FUNCTION_BLOCK FB_XPlanarModule EXTENDS FB_PackML_BaseModule
VAR
	// Component definitions here
	XPlanarTable : FB_Component_Xplanar := (Name := 'XPlanarTable');

	//Station Components
	Station1 : FB_RotateStation := (Name := 'Station1'); //Declaration of a custom station
	Station2 : FB_TiltStation := (Name := 'Station2');
	Station3 : FB_BounceStation := (Name := 'Station3');

	//Helper Vars
	Mover			  : ARRAY[1..SystemParameters.MOVER_COUNT] OF FB_XPlanarMover;
	Track			  : ARRAY[1..SystemParameters.TRACK_COUNT] OF FB_XPlanarTrackSegment;
	TracksInitialized : BOOL;
END_VAR

VAR_OUTPUT
	DCBusOK	: BOOL;
END_VAR

//! @summary This method contains code which will execute when this PackML module is in the <b>Aborting</b> state
METHOD PROTECTED Aborting
VAR
	i				: UDINT;
	SubModulesReady : BOOL := TRUE;
END_VAR
CASE DescendantSequenceState OF
	0:
		NoStateTasksToComplete := FALSE;
		NextStep(DescendantSequenceState);

	10:
		IF XPlanarTable.Abort() THEN
			StateTasksComplete := TRUE;
			NextStep(DescendantSequenceState);
		END_IF

	20:
		StateTasksComplete := TRUE;
END_CASE

SUPER^.Aborting();
END_METHOD

//! @summary This method contains code which will execute when this PackML module is in the <b>Clearing</b> state
METHOD PROTECTED Clearing
VAR
	i				: UDINT;
	SubModulesReady : BOOL := TRUE;
END_VAR

VAR_INST
	ipResult : I_PlanarTaskResult;
END_VAR

(*! <description> <b>Note:</b> The <i>Clear</i> command can also be thought of as a <i>fault reset</i> depite the ambiguity in the naming of the <i>Reset</i> state. 
<table> 
	<tr>
		<th> Previous State </th>
		<th> Transition In </th>
		<th> Transition Out </th>
		<th> Next State  </th> 
	</tr>
	<tr>
		<td> Aborted </td>
		<td> Clear Command </td> 
		<td> State Complete </td>
		<td> Stopped </td> 
	</tr>
</table>
This method is called as required by <c>StateControl()</c>
</description> 

*)
CASE _CurrentMode OF
	E_PMLUnitMode.ePMLUnitMode_Production:
		CASE DescendantSequenceState OF
			0: //Init
				NoStateTasksToComplete := FALSE;

				//Reset Stations
				Station1.Reset();
				Station2.Reset();
				Station3.Reset();
				
				XPlanarTable._Error		:= FALSE;
				XPlanarTable._ErrorID	:= 0;
					
				NextStep(DescendantSequenceState);

			10: //Reset XPlanar System
				IF XPlanarTable.Reset() THEN
					NextStep(DescendantSequenceState);
				END_IF

			20: //Enable Group
				ipResult := XPlanarTable.EnableGroup();
				IF ipResult.Done THEN
					NextStep(DescendantSequenceState);
				ELSIF ipResult.Error THEN
					ErrorStep(DescendantSequenceState);
				END_IF
				
			30:	// Re-detect movers
				ipResult	:= XPlanarTable.MoverRedetect();
				IF ipResult.Done THEN
					NextStep(DescendantSequenceState);
				ELSIF ipResult.Error THEN
					ErrorStep(DescendantSequenceState);
				END_IF

			40: //Clearing complete			
				StateTasksComplete := TRUE;
		END_CASE

	E_PMLUnitMode.ePMLUnitMode_Manual:
		;
END_CASE

SUPER^.Clearing();
END_METHOD

METHOD CyclicLogic
VAR
	i : INT;
END_VAR
IF NOT _InitComplete THEN
	_InitComplete := Initialize();
END_IF

//Call the base logic
SUPER^.CyclicLogic();
END_METHOD

//! @summary This method contains code which will execute when this PackML module is in the <b>Execute</b> state
METHOD PROTECTED Execute
VAR
	i : UDINT;
END_VAR
CASE _CurrentMode OF
	E_PMLUnitMode.ePMLUnitMode_Production:
		FOR i := 1 TO SystemParameters.STATION_COUNT DO
			ip.Stations[i].Execute();
		END_FOR

	E_PMLUnitMode.ePMLUnitMode_Manual:
		; //Insert logic for Manual Mode here
END_CASE
END_METHOD

//! @summary Automatically enables and disables HMI control based on the PackML mode
METHOD PROTECTED HMIPermissions

//! @description This method is called cyclically by <c>CyclicLogic()</c>
//General Mode Based Monitoring and handling of HMI control
CASE _CurrentMode OF
	E_PMLUnitMode.ePMLUnitMode_Production:
		AllowHMIControl(ThisModuleOnly := FALSE);

	E_PMLUnitMode.ePMLUnitMode_Manual:
		AllowHMIControl(ThisModuleOnly := FALSE);

	E_PMLUnitMode.ePMLUnitMode_Maintenance:
		AllowHMIControl(ThisModuleOnly := FALSE);
END_CASE
END_METHOD

//! @summary Basic module initialization logic
METHOD PROTECTED Initialize : BOOL;
VAR
	i						 : UDINT;
	varInfo					 : __SYSTEM.VAR_INFO;
	AllSubUnitsInitialized	 : BOOL := TRUE;
	AllComponentsInitialized : BOOL := TRUE;
END_VAR

//! @description This method is called by <c>CyclicLogic()</c> as required
Initialize := FALSE;
CASE DescendantSequenceState OF
	0: //Register Submodules and Components
		RegisterComponent(XPlanarTable);
		RegisterComponent(Station1);
		RegisterComponent(Station2);
		RegisterComponent(Station3);
		_LogModeChanges			:= FALSE;
		_LogStateChanges		:= FALSE;
		DescendantSequenceState := DescendantSequenceState + 10;

	10: //Set interfaces *This must be done before initializing the base class!

		//Set mover interfaces
		FOR i := 1 TO SystemParameters.MOVER_COUNT DO
			Mover[i].MoverIndex := i;
			ip.Movers[i]		:= Mover[i];
		END_FOR

		//Set Track Interfaces
		FOR i := 1 TO SystemParameters.TRACK_COUNT DO
			ip.Tracks[i] := Track[i];
		END_FOR

		//Set Station interfaces
		ip.Stations[1]			:= Station1;
		ip.Stations[2]			:= Station2;
		ip.Stations[3]			:= Station3;
		DescendantSequenceState := DescendantSequenceState + 10;

	20: //Call Initialize of the base class
		IF SUPER^.Initialize() THEN
			DescendantSequenceState := DescendantSequenceState + 10;
		END_IF

	30:
		Initialize := TRUE;
END_CASE
END_METHOD

METHOD PROTECTED Resetting
VAR_INST
	i			 : UDINT;
	ipTaskResult : I_PlanarTaskResult;
END_VAR
CASE _CurrentMode OF
	E_PMLUnitMode.ePMLUnitMode_Production:
		CASE DescendantSequenceState OF
			0: //Init
				i					   := 1;
				NoStateTasksToComplete := FALSE;
				NextStep(DescendantSequenceState);

			10: //Enable Tracks
				ipTaskResult := XplanarTable.EnableTracks();
				IF ipTaskResult.Done THEN
					NextStep(DescendantSequenceState);
				ELSIF ipTaskResult.Error THEN //An error occured, jump to 'error step'
					ErrorStep(DescendantSequenceState);
				END_IF

			20: //Enable Movers
				ipTaskResult := XPlanarTable.EnableMovers();
				IF ipTaskResult.Done THEN
					NextStep(DescendantSequenceState);
				ELSIF ipTaskResult.Error THEN //An error occured, jump to 'error step'
					ErrorStep(DescendantSequenceState);
				END_IF

			30: //Add Tracks to Group
				ipTaskResult := XPlanarTable.AddTracksToGroup();
				IF ipTaskResult.Done THEN
					NextStep(DescendantSequenceState);
				ELSIF ipTaskResult.Error THEN //An error occured, jump to 'error step'
					ErrorStep(DescendantSequenceState);
				END_IF

			40: //Add Movers to Group			
				ipTaskResult := XPlanarTable.AddMoversToGroup();
				IF ipTaskResult.Done THEN
					NextStep(DescendantSequenceState);
				ELSIF ipTaskResult.Error THEN //An error occured, jump to 'error step'
					ErrorStep(DescendantSequenceState);
				END_IF

			50: //Clearing complete
				StateTasksComplete := TRUE;
		END_CASE
END_CASE

SUPER^.Resetting();
END_METHOD

METHOD PRIVATE SetupStations : BOOL
VAR_INPUT
END_VAR
//Set Required Process Station Initialization Parameters
Station1.Position.SetValuesXYC(360, 120, 0);
Station1.Size.x		   := 120;		//Changes the station size in the X plane (optional - Default is 120mm)
Station1.Size.y		   := 120;		//Changes the station size in the Y plane (optionsl- Default is 120mm)
Station1.TrackID	   := 1;		//Set Index of the track segment the station resides on if applicable	
Station1.NextStation   := Station2; //Set the interface for the next station of the mover
Station1.StationAngle  := 180;
Station1.NumberOfTurns := 2;

Station2.Position.SetValuesXYC(120, 360, 0);
Station2.TrackID	   := 1;
Station2.NextStation   := Station3;
Station2.StationAngle  := 3.0;

Station3.Position.SetValuesXYC(360, 600, 0);
Station3.TrackID	   := 1;
Station3.NextStation   := Station1;
Station3.StationAngle  := -90;

//Return TRUE when all necessary station parameters are set
SetupStations := TRUE;
END_METHOD

METHOD PROTECTED Starting
VAR_INST
	i		 	: UDINT;
	ipResult 	: I_PlanarTaskResult;
	InitTimer	: TON;
END_VAR
CASE _CurrentMode OF
               E_PMLUnitMode.ePMLUnitMode_Production:
                              CASE DescendantSequenceState OF
                                             0:
                                                            NoStateTasksToComplete          := FALSE;
                                                            DescendantSequenceState      := 10;
                                                            i                                                           := 1;

                                             10: //Set Station Parameters
                                                            SetupStations();
                                                            NextStep(DescendantSequenceState);

                                             20: //Cleanup mover queues
                                                            FOR i := 1 TO SystemParameters.STATION_COUNT DO
                                                                           ip.Stations[i].MoverQueue.Dequeue();
                                                            END_FOR

                                                            NextStep(DescendantSequenceState);

                                             30: //Set some initial application move dynamics
                                                            FOR i := 1 TO SystemParameters.MOVER_COUNT DO
                                                                           ip.Movers[i].Dynamics.Movement.Accel             := 2000;
                                                                           ip.Movers[i].Dynamics.Movement.Decel            := 2000;
                                                                           ip.Movers[i].Dynamics.Movement.Velocity        := 300;
                                                                           ip.Movers[i].Dynamics.Movement.Jerk                := 50000;
                                                                           ip.Movers[i].Dynamics.Rotation.Accel                 := 5000;
                                                                           ip.Movers[i].Dynamics.Rotation.Decel                := 5000;
                                                                           ip.Movers[i].Dynamics.Rotation.Velocity            := 300;
                                                                           ip.Movers[i].Dynamics.Rotation.Jerk                    := 100000;
                                                                           ip.Movers[i].Dynamics.Tilt.Accel                            := 5000;
                                                                           ip.Movers[i].Dynamics.Tilt.Decel                            := 5000;
                                                                           ip.Movers[i].Dynamics.Tilt.Velocity                        := 300;
                                                                           ip.Movers[i].Dynamics.Tilt.Jerk                               := 100000;
                                                                           ip.Movers[i].Gap                                                           := 300;
                                                                           ip.Movers[i].Destination                                            := 0;
                                                            END_FOR

                                                            i := 1;
                                                            NextStep(DescendantSequenceState);
                                                            
                                             40: //Square Up movers
                                                            IF i <= SystemParameters.MOVER_COUNT THEN
                                                                           ipResult := ip.Movers[i].MoveCommand.SquareUp();
                                                                           IF ipResult.Done THEN
                                                                                          NextMinorStep(DescendantSequenceState);
                                                                           ELSIF ipResult.Error THEN
                                                                                          ErrorStep(DescendantSequenceState);
                                                                           END_IF
                                                            ELSE
                                                                           i := 1;
                                                                           NextStep(DescendantSequenceState);
                                                            END_IF                                              

                                             41: //Check Mover Count
                                                            IF i <= SystemParameters.MOVER_COUNT THEN
                                                                           I := i + 1;
                                                                           DescendantSequenceState := 40;
                                                            ELSE
                                                                           i := 1;
                                                                           NextStep(DescendantSequenceState);
                                                            END_IF
                                                            
                                             50: //Join Movers to nearest track
                                                            IF i <= SystemParameters.MOVER_COUNT THEN
                                                                           ipResult := ip.Movers[i].MoveCommand.JoinClosestTrack(FALSE);
                                                                           IF ipResult.Done THEN
                                                                                          NextMinorStep(DescendantSequenceState);
                                                                           ELSIF ipResult.Error THEN
                                                                                          ErrorStep(DescendantSequenceState);
                                                                           END_IF
                                                            ELSE
                                                                           i := 1;
                                                                           NextStep(DescendantSequenceState);
                                                            END_IF

                                             51: //Check Mover Count
                                                            IF i <= SystemParameters.MOVER_COUNT THEN
                                                                           I := i + 1;
                                                                           DescendantSequenceState := 50;
                                                            ELSE
                                                                           i := 1;
                                                                           NextStep(DescendantSequenceState);
                                                            END_IF

                                             60: //Send Movers around to station 1
                                                            IF i <= SystemParameters.MOVER_COUNT THEN
                                                                           ipResult := ip.Movers[i].MoveCommand.SendToStation(ip.Stations[1]);
                                                                           IF ipResult.Busy THEN
                                                                                          NextMinorStep(DescendantSequenceState);
                                                                           ELSIF ipResult.Error THEN
                                                                                          ErrorStep(DescendantSequenceState);
                                                                           END_IF
                                                            ELSE
                                                                           i := 1;
                                                                           NextStep(DescendantSequenceState);
                                                            END_IF

                                             61: //Check Mover Count
                                                            IF i <= SystemParameters.MOVER_COUNT THEN
                                                                           I := i + 1;
                                                                           DescendantSequenceState := 60;
                                                            ELSE
                                                                           i := 1;
                                                                           NextStep(DescendantSequenceState);
                                                            END_IF

                                             70: //Let recovery get moving before jumping to execute
                                                            InitTimer(IN := TRUE, PT := T#1000MS);
                                                            IF InitTimer.Q THEN
                                                                           InitTimer(IN := FALSE);
                                                                           StateTasksComplete := TRUE;
                                                            END_IF                
                              END_CASE

               E_PMLUnitMode.ePMLUnitMode_Manual:
                              ;
END_CASE

SUPER^.Starting();
END_METHOD

END_FUNCTION_BLOCK

(* stored: Version 1.1.0.1, ProductVersion 3.1.4024.13
   POU FB_XPlanarModule: Id {18ed3aa7-c83f-44ce-8119-20fe14cb0cfa}, SpecialFunc None
   Folder I_CyclicFB: Id {769d746d-1ab5-4a6d-8c77-4b1403733257}
   Folder Methods: Id {1414b749-8a1b-4539-8751-a9eb98ce9efa}
   Folder Acting States: Id {f6cfc130-33f5-4b9c-9ed3-b6e57724e54f}
   Folder HMI: Id {0f08a4f8-e768-454b-a528-0661effe207e}
   Folder Waiting States: Id {ab86d3ba-50da-471d-864b-21041ca20d53}
   Method Aborting: Id {17e4bd4f-b401-48a2-abdb-1c82c9b91958}
   Method Clearing: Id {749d9d49-762f-4674-b533-d711fd25e786}
   Method CyclicLogic: Id {31fa8ff0-2b84-4416-a54a-15ba032d89ac}
   Method Execute: Id {4a8447c7-4bba-456b-ae99-02b9655bd430}
   Method HMIPermissions: Id {7d2cddec-eedc-414c-8c02-c97cb122267e}
   Method Initialize: Id {cea669eb-9427-49e9-a099-b64514cc633b}
   Method Resetting: Id {31624805-9f24-4846-bb15-1edf775cd7f4}
   Method SetupStations: Id {472d87c4-f8ee-4679-a5bf-c6f2e3004197}
   Method Starting: Id {183f1123-c447-4a86-b202-a4cab71a6c14} *)
